RESOURCE_TYPE topFLAT
  (* Standard: 61499-2 *)
  (* Version 0.1, 2017-00-09, Hammond, HAMMONDSDESKTOP *)
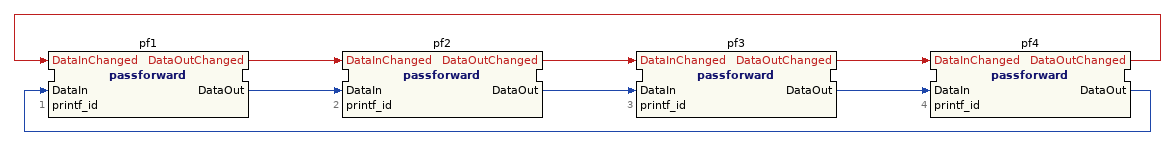
  FBS
    pf1 : passforward(printf_id := 1);
    pf2 : passforward(printf_id := 2);
    pf3 : passforward(printf_id := 3);
    pf4 : passforward(printf_id := 4);
  END_FBS
  EVENT_CONNECTIONS
    pf1.DataOutChanged TO pf2.DataInChanged;
    pf2.DataOutChanged TO pf3.DataInChanged;
    pf3.DataOutChanged TO pf4.DataInChanged;
    pf4.DataOutChanged TO pf1.DataInChanged;
  END_CONNECTIONS
  DATA_CONNECTIONS
    pf1.DataOut TO pf2.DataIn;
    pf2.DataOut TO pf3.DataIn;
    pf3.DataOut TO pf4.DataIn;
    pf4.DataOut TO pf1.DataIn;
  END_CONNECTIONS
END_RESOURCE_TYPE
